// TIA Portal V19 export
DATA_BLOCK "TRCV_DI"   // DB367
// stored: AutoNumber false, InstanceOfName TRCV, OfSystemLibElement TRCV, OfSystemLibVersion 4.0
"TRCV"
   // VAR_INPUT
   //    EN_R : Bool := TRUE;
   //    ID : CONN_OUC := 16#0002;
   //    LEN : UDInt := 30;
   //    ADHOC : Bool := FALSE;
   // END_VAR
   // VAR_OUTPUT
   //    NDR : Bool := TRUE;
   //    BUSY : Bool := FALSE;
   //    ERROR : Bool := FALSE;
   //    STATUS : Word := 16#0000;
   //    RCVD_LEN : UDInt := 30;
   // END_VAR
   // VAR_IN_OUT
   //    DATA : Variant;
   //    ADDR : Variant;
   // END_VAR
BEGIN
END_DATA_BLOCK
